{attribute addProperty BoxType "EK1122-0000-0018"}
{attribute addProperty Id "Beckhoff_EJ4xxxsub_EK1100EK1100_179A0949162"}
{attribute addProperty CRC "363478827"}
{attribute addProperty SizeInBites "16"}
{attribute addProperty SizeInBytes "2"}
TYPE Beckhoff_EJ4xxxEK1122_15AA3F2B EXTENDS EK1122_179A0949 :
STRUCT
	{attribute addProperty Name "Beckhoff_EJ4xxxsub_EK1100"}
	Beckhoff_EJ4xxxsub_EK1100 : EK1100_179A0949;
END_STRUCT
END_TYPE

(* stored: Version 1.2.0.0, ProductVersion 3.1.4024.9
   DUT Beckhoff_EJ4xxxEK1122_15AA3F2B: Id {5a4fc442-f585-4556-a758-80f85af2c8da} *)
